FUNCTION_BLOCK ALU (* Template for a simple Basic Function Block Type *)
  (* Standard: 61499-2 *)
  (* Version 1.0, 2020-12-24, jetbrains *)
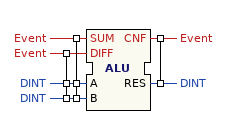
  EVENT_INPUT
    SUM WITH A, B; (* Event inputs *)
    DIFF WITH A, B;
  END_EVENT
  EVENT_OUTPUT
    CNF WITH RES; (* Execution Confirmation *)
  END_EVENT
  VAR_INPUT
    A : DINT; (* Input event qualifier *)
    B : DINT;
  END_VAR
  VAR_OUTPUT
    RES : DINT; (* Output event qualifier *)
  END_VAR
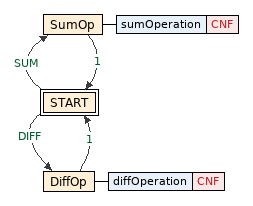
  EC_STATES
    START; (* Initial State *)
    SumOp : sumOperation -> CNF; (* Normal execution *)
    DiffOp : diffOperation -> CNF;
  END_STATES
  EC_TRANSITIONS
    START TO SumOp := SUM;
    SumOp TO START := 1;
    START TO DiffOp := DIFF;
    DiffOp TO START := 1;
  END_TRANSITIONS
  ALGORITHM sumOperation IN ST: (* new algorithm *)
RES := A + B;
  END_ALGORITHM
  ALGORITHM diffOperation IN ST:
RES := A - B;
  END_ALGORITHM
END_FUNCTION_BLOCK
